// Convert analog value to normalized value
FUNCTION AnalogInputConversion : REAL
VAR_INPUT
	// Analog Value to normalize
	AnalogInput : WORD;
	// Maximum value on the scale
	ScaleMax: INT;
END_VAR
VAR
	NormalizedInput: REAL;
END_VAR

VAR_OUTPUT
	// Normalized Output
	ScaledValue: REAL;
END_VAR

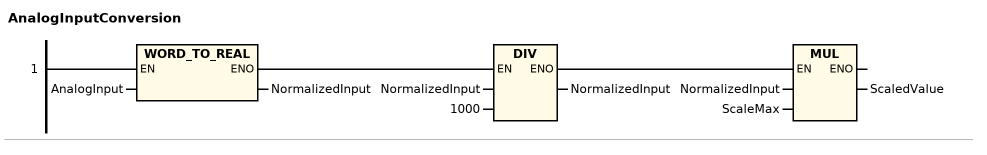
// NETWORK 1
NormalizedInput := WORD_TO_REAL(AnalogInput);
NormalizedInput := NormalizedInput / 1000;
ScaledValue := NormalizedInput * ScaleMax;

END_FUNCTION

(* stored: Version 1.1.0.1, ProductVersion 3.1.4024.12
   POU AnalogInputConversion: Id {378ca282-7c72-4964-ba91-45d6b7fec8b6}, SpecialFunc None *)
